Fanuc KAREL source: kt00025.KL

-- PROVISIONAL review KL for V1013-1; original PC SHA256 24caef9cc6e3c3fe28509fb9108b9023e9c6ed3ccbb23c6359abc2c66ce7bd01
-- Incomplete behavior may be omitted. Consult companion uncertainty JSON. Do not deploy.
PROGRAM KT00025
%NOLOCKGROUP
VAR
  I2 : INTEGER
  OUT : INTEGER
-- UNRESOLVED_DECL H1 type=002017
BEGIN
  -- UNRESOLVED_PC offsets 5-19; opcodes 2E,22,9D,33,B4
  -- UNRESOLVED_PC offsets 24-35; opcodes 2E,23
  -- UNRESOLVED_PC offsets 40-62; opcodes 22,9D,33,B3,21,52,23
  -- UNRESOLVED_PC offsets 67-71; opcodes 7F
END KT00025
